Staubli VAL3: setSamPosOffs.pgx

program setSamPosOffs(string inputMessage, num sio_ID)
  local bool isNumber[2]
  local bool isOK
  local num msgLength
  local string reply
  local pointRx samplePosPnt
  local num xMsgIndex
  local num yMsgIndex
begin
  //**************************************************
  // Method to set the coordinates of currentSamPosj (current sample position).
  // Messages take the form:
  //     setSamPosOffset:#X1#Y2
  // Coordinate system starts at 0 (e.g. X=0, Y=0 is first sample position)
  //**************************************************

  // To start with the function is assumed working and we print the input
  isOK=true
  putln("Setting magazine coordinates:")
  putln("   "+inputMessage)

  // Find the where the coordinates are being supplied
  xMsgIndex=find(inputMessage,"#X")
  yMsgIndex=find(inputMessage,"#Y")
  msgLength=len(inputMessage)

  // Extract the numSamPos from the message and convert string to number
  toNum(mid(inputMessage,(yMsgIndex-(xMsgIndex+2)),(xMsgIndex+2)),numSamOffs[0],isNumber[0])
  toNum(mid(inputMessage,(msgLength-(yMsgIndex+2)),(yMsgIndex+2)),numSamOffs[1],isNumber[1])

  // Check conversion to number successful and print to screen
  isOK=isOK and isNumber[0] and isNumber[1]
  if isNumber[0]==false
    reply="setSamPos:fail_'Invalid X'"
    put("Failed setting X. Found: ")
    putln(right(inputMessage,(yMsgIndex-(xMsgIndex+2))))
  elseIf isNumber[1]==false
    reply="setSamPos:fail_'Invalid Y'"
    put("Failed setting Y. Found: ")
    putln(right(inputMessage,(msgLength-(yMsgIndex+2))))
  endIf

  // Assuming we got the numbers, now we create our new joint coordinate
  if isOK==true
    put("SamPos: X=")
    put(numSamOffs[0])
    put(" Y=")
    putln(numSamOffs[1])
    samplePosPnt=appro(jointToPoint(flange,world,homePosition),{(numSamOffs[0])*-17.03,(numSamOffs[1])*-17,0,0,0,0})
    isOK=pointToJoint(flange,homePosition,samplePosPnt,currentSamPosJ)

    // Update knownPositions collection
    knownPositions["currentSamPos"] = currentSamPosJ

    if isOK==true
      reply="setSamPosOffset:done"
    else
      reply="setSamPosOffset:fail_'Could not convert position to joint'"
      putln("Failed converting position to joint")
    endIf
  endIf

  taskCreate "sendStatus",10,sendStatus(reply,sio_ID)
  taskKill("setSamPosOffset")
end
